FUNCTION_BLOCK FB_Hmi_Switch EXTENDS FB_Hmi_Component
VAR
	_rSwitch: REFERENCE TO S_Hmi_Switch;
END_VAR

IF _initialized THEN
	IF _rSwitch.Click THEN
		Toggle();
	END_IF
END_IF

_rSwitch.Click := FALSE;

PROPERTY PUBLIC Enabled : BOOL
SET
_rSwitch.Enabled := Enabled;
END_SET
END_PROPERTY

METHOD PUBLIC Initialize : BOOL
VAR_INPUT
	rSwitch: REFERENCE TO S_Hmi_Switch;
END_VAR
IF __ISVALIDREF(rSwitch) THEN
	_rSwitch REF= rSwitch;

	_initialized := Initialize := TRUE;
END_IF
END_METHOD

METHOD PUBLIC Reset
IF _initialized AND_THEN _rSwitch.Enabled THEN
	_rSwitch.Value := FALSE;
END_IF
END_METHOD

METHOD PUBLIC Set
IF _initialized AND_THEN _rSwitch.Enabled THEN
	_rSwitch.Value := TRUE;
END_IF
END_METHOD

METHOD PUBLIC Toggle
IF _initialized AND_THEN _rSwitch.Enabled THEN
	_rSwitch.Value := NOT _rSwitch.Value;
END_IF
END_METHOD

PROPERTY PUBLIC Value : BOOL
GET
Value := _rSwitch.Value;
END_GET
END_PROPERTY

PROPERTY PUBLIC Visibility : BOOL
SET
IF _initialized THEN
	_rSwitch.Visibility := Visibility;
END_IF
END_SET
END_PROPERTY

END_FUNCTION_BLOCK

(* stored: Version 1.1.0.1, ProductVersion 3.1.4024.10
   POU FB_Hmi_Switch: Id {88713cc5-8b82-46e1-8462-6e1bd39a71c9}, SpecialFunc None
   Property Enabled: Id {e7726983-7a03-4966-b733-88091e0634c4}
   Set Set: Id {9dc6da4a-5294-469e-a003-543fcf8ab797}
   Method Initialize: Id {559c6346-41d8-460b-a26e-b14f3b23b94d}
   Method Reset: Id {17ed8b5e-134b-4111-b89b-b4755b9d56b7}
   Method Set: Id {b83c55f3-9c64-4f44-8441-dfa045eac25c}
   Method Toggle: Id {6bd9f366-31f1-4de6-9e3c-2c0e9b172c9e}
   Property Value: Id {51018a77-834b-4386-b410-1383627bc519}
   Get Get: Id {5e522851-3fdc-44d2-960e-9819d53b6bcd}
   Property Visibility: Id {a35c6be8-c610-4450-822a-8a50b51090f8}
   Set Set: Id {13fe9c60-01b0-461e-a814-c8e63448beb7} *)
